FUNCTION_BLOCK FB_CommandChangeUnHold EXTENDS FB_CommandChange IMPLEMENTS ITF_CommandChange
VAR

END_VAR

(*			
	EVERDE sp. z o.o.
	Rafał Osajda		03.11.2025		TC 4024.66
	Test czy można zmienić stan lub tryb i zwraca czy można i uruchamia zmianę
*)
METHOD PUBLIC Execute : BOOL
VAR_INPUT
END_VAR
IF (TRUE) THEN
	THIS^.itfSaMController.ChangeStateTo (eNewState := E_SaMStates.Unholding);
END_IF
END_METHOD

METHOD FB_init : BOOL
VAR_INPUT
	bInitRetains : BOOL; // if TRUE, the retain variables are initialized (warm start / cold start)
	bInCopyCode : BOOL;  // if TRUE, the instance afterwards gets moved into the copy code (online change)
END_VAR
THIS^.SetText (eLocation := E_BaseLocation.pl, wsDescription := "Command change state - UnHold");
THIS^.SetText (eLocation := E_BaseLocation.en, wsDescription := "Command change state - UnHold");
THIS^.SetText (eLocation := E_BaseLocation.de, wsDescription := "Command change state - UnHold");
THIS^.SetName (stName := THIS^.GetTexts ());
END_METHOD

END_FUNCTION_BLOCK

(* stored: Version 1.1.0.1
   POU FB_CommandChangeUnHold: Id {2192cb93-53a7-0597-0430-86ec6d252e43}, SpecialFunc None
   Method Execute: Id {acc076f0-f8b5-0918-2baf-caffadaef7de}
   Method FB_init: Id {d9be5a9a-d672-06ae-1396-1299af8de0a3} *)
